FUNCTION_BLOCK FB_SimCheckWeigher
VAR_INPUT
END_VAR
VAR_OUTPUT
END_VAR
VAR
	bLift						AT %I* : BOOL;
	fScaleReading				AT %Q* : LREAL;
	bPartPresent				AT %Q* : BOOL;
	
	rand						: DRAND;
	fWeightSetpoint				: LREAL := 1000.0;
	tmrWork						: TON;
	iWorkMs						: DINT;
	iState						: DINT;
END_VAR

rand(Seed:=MAIN.Seed+13);

CASE iState OF
	0:
		IF bLift THEN
			iState := 10;
		ELSE
			fScaleReading := 0.0 + (rand.Num / 5000);
		END_IF

	10:
		IF fScaleReading < fWeightSetpoint THEN
			fScaleReading := fScaleReading + (fWeightSetpoint / 50) + (rand.Num * 10);
		ELSE
			iState := 20;
		END_IF
		
	20:
		IF bLift THEN
			IF fScaleReading < fWeightSetpoint THEN
				fScaleReading := fScaleReading + rand.Num;
			ELSE
				fScaleReading := fScaleReading - rand.Num;
			END_IF
		ELSE
			iState := 0;
		END_IF
		
END_CASE

PROPERTY PUBLIC PartPresent : BOOL
GET
PartPresent := bPartPresent;
END_GET
SET
bPartPresent := PartPresent;
END_SET
END_PROPERTY

END_FUNCTION_BLOCK

(* stored: Version 1.1.0.1, ProductVersion 3.1.4024.12
   POU FB_SimCheckWeigher: Id {92bab77b-be28-48d9-9ba6-55ffa9050dd6}, SpecialFunc None
   Property PartPresent: Id {0d2531d8-1940-42c4-b0c2-849dfc637b41}
   Get Get: Id {89580202-1e1c-4436-b39d-e116d591c4bc}
   Set Set: Id {1aa9f137-4566-4a00-8fbd-3af25d42fcc4} *)
